TYPE uWORD_BOOL_MX2 :
UNION
	bits 			:ARRAY [0..15] OF BOOL;
	ch 				:WORD;
	
END_UNION
END_TYPE

(* stored: Version 1.1.0.1, ProductVersion 3.1.4022.12
   DUT uWORD_BOOL_MX2: Id {d4fffac4-f061-468b-898e-ecaef371cfd4} *)
